// Provides basic string builder implementation
FUNCTION_BLOCK FB_StringBuilderBase IMPLEMENTS I_StringBuilder;
VAR
	_string	: Tc2_System.T_MaxString;
END_VAR

(* Adds a string to the build sequence.*)
METHOD AddString : I_StringBuilder
VAR_INPUT
	(* String to be added.*)
	str	: Tc2_System.T_MaxString;
END_VAR
_string := Tc2_Standard.CONCAT(
	STR1 := _string, 
	STR2 := str);
	
AddString := THIS^;
END_METHOD

(* Finishes string generation and returns the generated string*)
METHOD Create : Tc2_System.T_MaxString
Create := _string;
END_METHOD

(* Reset the string build sequence, clear any string built so far.*)
METHOD Reset : I_StringBuilder
_string := '';
Reset := THIS^;
END_METHOD

END_FUNCTION_BLOCK

(* stored: Version 1.1.0.1, ProductVersion 3.1.4024.13
   POU FB_StringBuilderBase: Id {4af2ae7b-34e5-0402-2ab5-b787ed381493}, SpecialFunc None
   Method AddString: Id {a1f2665a-9e23-0057-3cb2-001019efbfb5}
   Method Create: Id {837ad951-dde3-0ecc-1e91-80edffc6563f}
   Method Reset: Id {c0b64bb0-ab5a-04e6-313f-3575f6a54110} *)
